{attribute 'linkalways'} 
{attribute 'no_explicit_call' := 'This FB is a CLASS and must be accessed using methods or properties'}
{attribute 'enable_dynamic_creation'}
FUNCTION_BLOCK INTERNAL ABSTRACT Mc2AxisCommand EXTENDS AsyncCommand IMPLEMENTS AxisCommand
VAR
	axis : Axis;
END_VAR

END_FUNCTION_BLOCK

(* stored: Version 1.1.0.1, ProductVersion 3.1.4026.13
   POU Mc2AxisCommand: Id {fd1615e8-bcb5-04fd-2c76-cb04779223d2}, SpecialFunc None *)
